FUNCTION_BLOCK L3_PartMerge (* Part adapter encapculation *)
  (* Standard: 61499-2; Description: This block is used to encapsulate all the events and data, used to manage the manufacturing of part, into an adapter. *)
  (* Version 0.0, 2014-09-24, EQUEROL, UJI *)
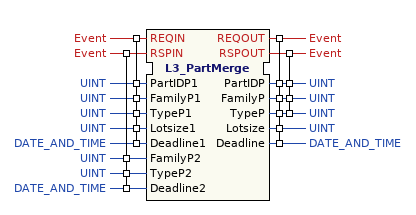
  EVENT_INPUT
    REQIN WITH FamilyP1, TypeP1, Lotsize1, Deadline1, PartIDP1; (* Normal Execution Request *)
    RSPIN WITH FamilyP2, TypeP2, Deadline2; (* Ended part reception confirmation *)
  END_EVENT
  EVENT_OUTPUT
    REQOUT WITH PartIDP, FamilyP, TypeP, Lotsize, Deadline; (* Execution Confirmation *)
    RSPOUT WITH PartIDP, FamilyP, TypeP; (* Ended part indication *)
  END_EVENT
  VAR_INPUT
    PartIDP1 : UINT; (* Identifier of the 1st part to be manufactured *)
    FamilyP1 : UINT; (* Part's family *)
    TypeP1 : UINT; (* Part's type *)
    Lotsize1 : UINT; (* Number of parts to be in the order *)
    Deadline1 : DATE_AND_TIME; (* Deadline of next part to be delivered *)
    FamilyP2 : UINT; (* Part's family *)
    TypeP2 : UINT; (* Part's type *)
    Deadline2 : DATE_AND_TIME; (* Deadline of next part to be delivered *)
  END_VAR
  VAR_OUTPUT
    PartIDP : UINT; (* Part identifier *)
    FamilyP : UINT; (* Part's family *)
    TypeP : UINT; (* Part's type *)
    Lotsize : UINT; (* Number of parts to be in the order *)
    Deadline : DATE_AND_TIME; (* Deadline of next part to be delivered *)
  END_VAR
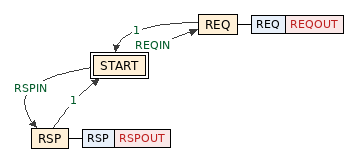
  EC_STATES
    START; (* Initial State *)
    REQ : REQ -> REQOUT; (* Normal execution *)
    RSP : RSP -> RSPOUT;
  END_STATES
  EC_TRANSITIONS
    START TO REQ := REQIN;
    REQ TO START := 1;
    START TO RSP := RSPIN;
    RSP TO START := 1;
  END_TRANSITIONS
  ALGORITHM REQ IN ST: (* Sends REQ event and data through the adapter *)
(*Map input data into the adapter*)
PartIDP := PartIDP1;
FamilyP := FamilyP1;
TypeP := TypeP1;
Lotsize := Lotsize1;
Deadline := Deadline1;
  END_ALGORITHM
  ALGORITHM RSP IN ST: (* Sends RSP event and data through the adapter *)
(*Map input data into the adapter*)
FamilyP := FamilyP2;
TypeP := TypeP2;
Deadline := Deadline2;
  END_ALGORITHM
END_FUNCTION_BLOCK
